// TIA Portal V21 export
FUNCTION "FC603" : Void   // FC603, LAD
TITLE = FC603
{ S7_Optimized_Access := 'TRUE' }
// CIP logic
// stored: AutoNumber false, SetENOAutomatically false
   VAR_TEMP
      temp : Int;
      re : Bool;
   END_VAR
   VAR_TEMP   // added for the SCL form of the ladder/FBD networks
      _w1 : Bool;
      _w2 : Bool;
      _w3 : Bool;
   END_VAR
BEGIN

REGION Network 1: NoCycleSelectedInterlock
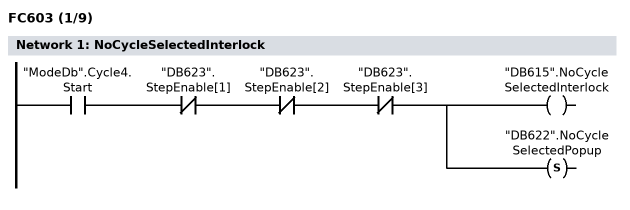
   RUNG wire#powerrail
      Contact( "ModeDb".Cycle4.Start )
      I_Contact( "DB623".StepEnable[1] )
      I_Contact( "DB623".StepEnable[2] )
      I_Contact( "DB623".StepEnable[3] )
      wire#w1
      Coil( "DB615".NoCycleSelectedInterlock )
   END_RUNG
   RUNG wire#w1
      S_Coil( "DB622".NoCycleSelectedPopup )
   END_RUNG
   // the same network as SCL:
   "DB615".NoCycleSelectedInterlock := "ModeDb".Cycle4.Start AND NOT "DB623".StepEnable[1] AND NOT "DB623".StepEnable[2] AND NOT "DB623".StepEnable[3];
   IF "DB615".NoCycleSelectedInterlock THEN "DB622".NoCycleSelectedPopup := TRUE; END_IF;
END_REGION

REGION Network 2: "DB615".Fault
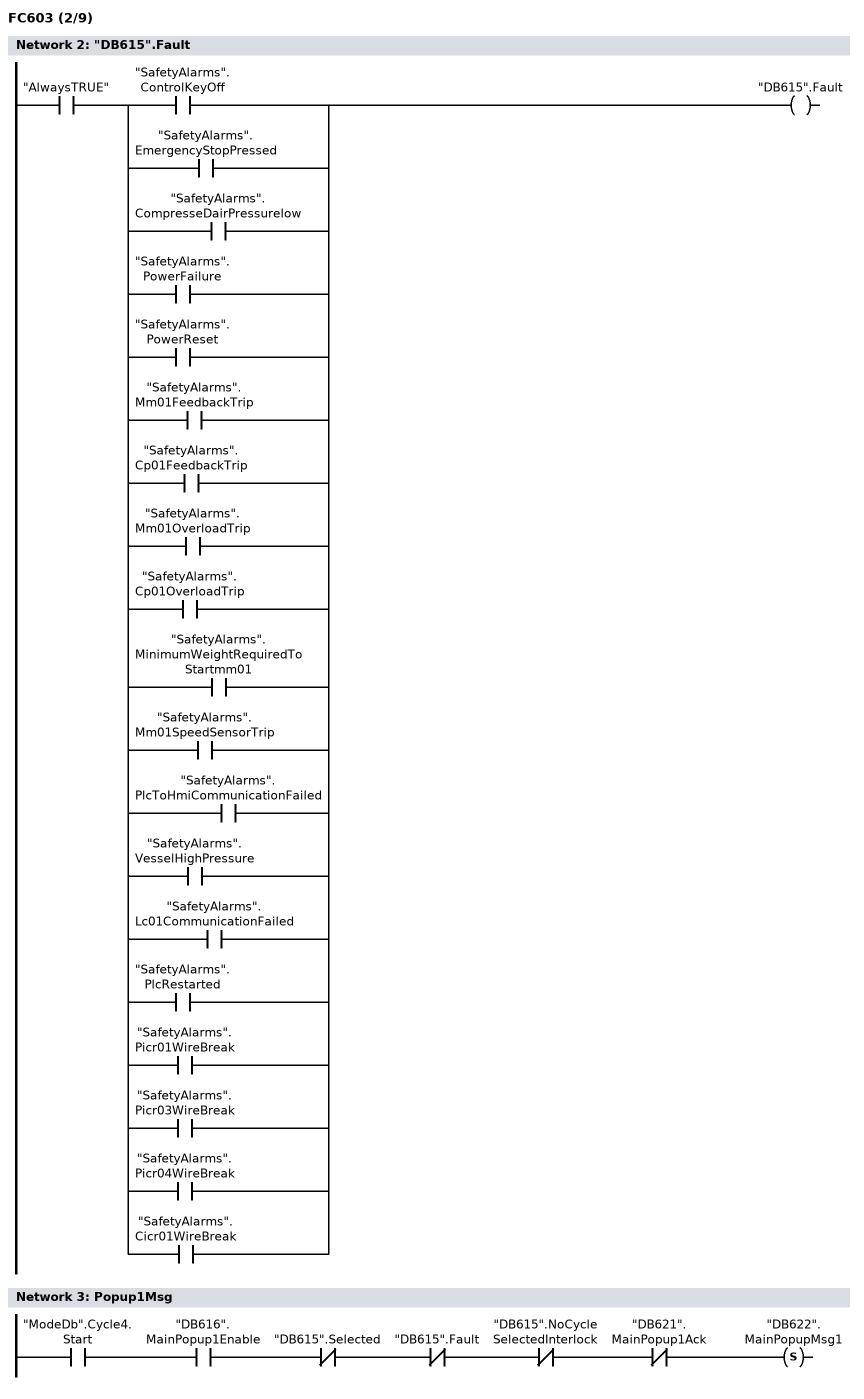
   RUNG wire#powerrail
      Contact( "AlwaysTRUE" )
      wire#w1
      Contact( "SafetyAlarms".ControlKeyOff )
      wire#w2
      Coil( "DB615".Fault )
   END_RUNG
   RUNG wire#w1
      Contact( "SafetyAlarms".EmergencyStopPressed )
   END_RUNG wire#w2
   RUNG wire#w1
      Contact( "SafetyAlarms".CompresseDairPressurelow )
   END_RUNG wire#w2
   RUNG wire#w1
      Contact( "SafetyAlarms".PowerFailure )
   END_RUNG wire#w2
   RUNG wire#w1
      Contact( "SafetyAlarms".PowerReset )
   END_RUNG wire#w2
   RUNG wire#w1
      Contact( "SafetyAlarms".Mm01FeedbackTrip )
   END_RUNG wire#w2
   RUNG wire#w1
      Contact( "SafetyAlarms".Cp01FeedbackTrip )
   END_RUNG wire#w2
   RUNG wire#w1
      Contact( "SafetyAlarms".Mm01OverloadTrip )
   END_RUNG wire#w2
   RUNG wire#w1
      Contact( "SafetyAlarms".Cp01OverloadTrip )
   END_RUNG wire#w2
   RUNG wire#w1
      Contact( "SafetyAlarms".MinimumWeightRequiredToStartmm01 )
   END_RUNG wire#w2
   RUNG wire#w1
      Contact( "SafetyAlarms".Mm01SpeedSensorTrip )
   END_RUNG wire#w2
   RUNG wire#w1
      Contact( "SafetyAlarms".PlcToHmiCommunicationFailed )
   END_RUNG wire#w2
   RUNG wire#w1
      Contact( "SafetyAlarms".VesselHighPressure )
   END_RUNG wire#w2
   RUNG wire#w1
      Contact( "SafetyAlarms".Lc01CommunicationFailed )
   END_RUNG wire#w2
   RUNG wire#w1
      Contact( "SafetyAlarms".PlcRestarted )
   END_RUNG wire#w2
   RUNG wire#w1
      Contact( "SafetyAlarms".Picr01WireBreak )
   END_RUNG wire#w2
   RUNG wire#w1
      Contact( "SafetyAlarms".Picr03WireBreak )
   END_RUNG wire#w2
   RUNG wire#w1
      Contact( "SafetyAlarms".Picr04WireBreak )
   END_RUNG wire#w2
   RUNG wire#w1
      Contact( "SafetyAlarms".Cicr01WireBreak )
   END_RUNG wire#w2
   // the same network as SCL:
   "DB615".Fault := "AlwaysTRUE" AND ("SafetyAlarms".ControlKeyOff OR "SafetyAlarms".EmergencyStopPressed OR "SafetyAlarms".CompresseDairPressurelow OR "SafetyAlarms".PowerFailure OR "SafetyAlarms".PowerReset OR "SafetyAlarms".Mm01FeedbackTrip OR "SafetyAlarms".Cp01FeedbackTrip OR "SafetyAlarms".Mm01OverloadTrip OR "SafetyAlarms".Cp01OverloadTrip OR "SafetyAlarms".MinimumWeightRequiredToStartmm01 OR "SafetyAlarms".Mm01SpeedSensorTrip OR "SafetyAlarms".PlcToHmiCommunicationFailed OR "SafetyAlarms".VesselHighPressure OR "SafetyAlarms".Lc01CommunicationFailed OR "SafetyAlarms".PlcRestarted OR "SafetyAlarms".Picr01WireBreak OR "SafetyAlarms".Picr03WireBreak OR "SafetyAlarms".Picr04WireBreak OR "SafetyAlarms".Cicr01WireBreak);
END_REGION

REGION Network 3: Popup1Msg
   RUNG wire#powerrail
      Contact( "ModeDb".Cycle4.Start )
      Contact( "DB616".MainPopup1Enable )
      I_Contact( "DB615".Selected )
      I_Contact( "DB615".Fault )
      I_Contact( "DB615".NoCycleSelectedInterlock )
      I_Contact( "DB621".MainPopup1Ack )
      S_Coil( "DB622".MainPopupMsg1 )
   END_RUNG
   // the same network as SCL:
   IF "ModeDb".Cycle4.Start AND "DB616".MainPopup1Enable AND NOT "DB615".Selected AND NOT "DB615".Fault AND NOT "DB615".NoCycleSelectedInterlock AND NOT "DB621".MainPopup1Ack THEN
       "DB622".MainPopupMsg1 := TRUE;
   END_IF;
END_REGION

REGION Network 4: Popup2Msg
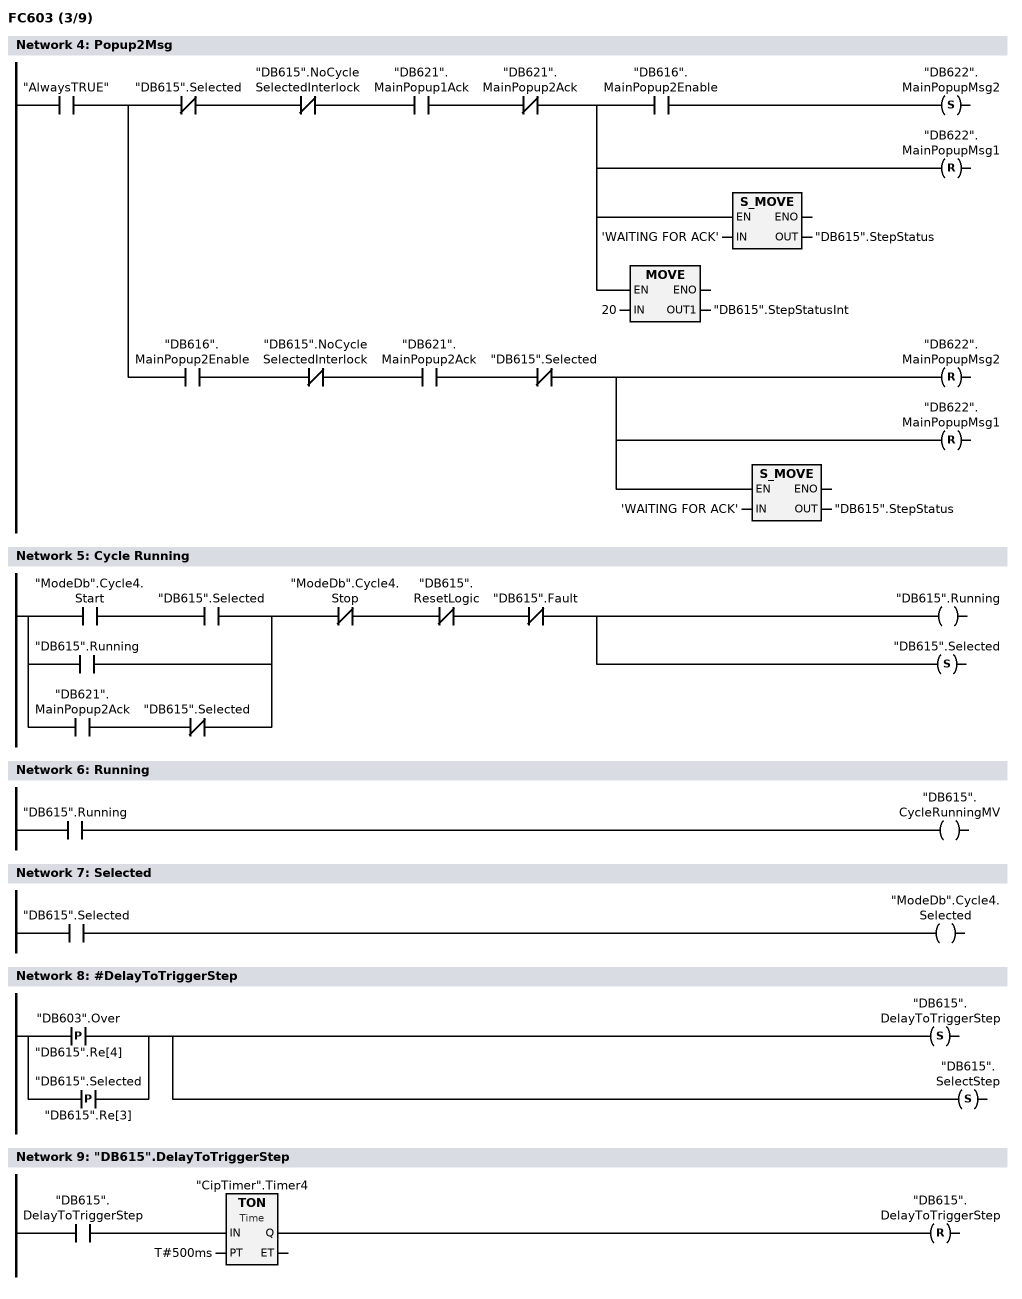
   RUNG wire#powerrail
      Contact( "AlwaysTRUE" )
      wire#w1
      I_Contact( "DB615".Selected )
      I_Contact( "DB615".NoCycleSelectedInterlock )
      Contact( "DB621".MainPopup1Ack )
      I_Contact( "DB621".MainPopup2Ack )
      wire#w2
      Contact( "DB616".MainPopup2Enable )
      S_Coil( "DB622".MainPopupMsg2 )
   END_RUNG
   RUNG wire#w2
      R_Coil( "DB622".MainPopupMsg1 )
   END_RUNG
   RUNG wire#w2
      S_Move(in := 'WAITING FOR ACK', out => "DB615".StepStatus)
   END_RUNG
   RUNG wire#w2
      Move(in := 20, out1 => "DB615".StepStatusInt)
   END_RUNG
   RUNG wire#w1
      Contact( "DB616".MainPopup2Enable )
      I_Contact( "DB615".NoCycleSelectedInterlock )
      Contact( "DB621".MainPopup2Ack )
      I_Contact( "DB615".Selected )
      wire#w3
      R_Coil( "DB622".MainPopupMsg2 )
   END_RUNG
   RUNG wire#w3
      R_Coil( "DB622".MainPopupMsg1 )
   END_RUNG
   RUNG wire#w3
      S_Move(in := 'WAITING FOR ACK', out => "DB615".StepStatus)
   END_RUNG
   // the same network as SCL:
   #_w1 := "AlwaysTRUE" AND NOT "DB615".Selected AND NOT "DB615".NoCycleSelectedInterlock AND "DB621".MainPopup1Ack AND NOT "DB621".MainPopup2Ack;
   IF #_w1 AND "DB616".MainPopup2Enable THEN "DB622".MainPopupMsg2 := TRUE; END_IF;
   IF #_w1 THEN
       "DB622".MainPopupMsg1 := FALSE;
       "DB615".StepStatus := 'WAITING FOR ACK';
       "DB615".StepStatusInt := 20;
   END_IF;
   IF "AlwaysTRUE" AND "DB616".MainPopup2Enable AND NOT "DB615".NoCycleSelectedInterlock AND "DB621".MainPopup2Ack AND NOT "DB615".Selected THEN
       "DB622".MainPopupMsg2 := FALSE;
       "DB622".MainPopupMsg1 := FALSE;
       "DB615".StepStatus := 'WAITING FOR ACK';
   END_IF;
END_REGION

REGION Network 5: Cycle Running
   RUNG wire#powerrail
      Contact( "ModeDb".Cycle4.Start )
      Contact( "DB615".Selected )
      wire#w1
      I_Contact( "ModeDb".Cycle4.Stop )
      I_Contact( "DB615".ResetLogic )
      I_Contact( "DB615".Fault )
      wire#w2
      Coil( "DB615".Running )
   END_RUNG
   RUNG wire#powerrail
      Contact( "DB615".Running )
   END_RUNG wire#w1
   RUNG wire#powerrail
      Contact( "DB621".MainPopup2Ack )
      I_Contact( "DB615".Selected )
   END_RUNG wire#w1
   RUNG wire#w2
      S_Coil( "DB615".Selected )
   END_RUNG
   // the same network as SCL:
   "DB615".Running := (("ModeDb".Cycle4.Start AND "DB615".Selected) OR "DB615".Running OR ("DB621".MainPopup2Ack AND NOT "DB615".Selected)) AND NOT "ModeDb".Cycle4.Stop AND NOT "DB615".ResetLogic AND NOT "DB615".Fault;
   IF "DB615".Running THEN "DB615".Selected := TRUE; END_IF;
END_REGION

REGION Network 6: Running
   RUNG wire#powerrail
      Contact( "DB615".Running )
      Coil( "DB615".CycleRunningMV )
   END_RUNG
   // the same network as SCL:
   "DB615".CycleRunningMV := "DB615".Running;
END_REGION

REGION Network 7: Selected
   RUNG wire#powerrail
      Contact( "DB615".Selected )
      Coil( "ModeDb".Cycle4.Selected )
   END_RUNG
   // the same network as SCL:
   "ModeDb".Cycle4.Selected := "DB615".Selected;
END_REGION

REGION Network 8: #DelayToTriggerStep
   RUNG wire#powerrail
      P_Contact(operand := "DB603".Over, bit := "DB615".Re[4])
      wire#w1
      S_Coil( "DB615".DelayToTriggerStep )
   END_RUNG
   RUNG wire#powerrail
      P_Contact(operand := "DB615".Selected, bit := "DB615".Re[3])
   END_RUNG wire#w1
   RUNG wire#w1
      S_Coil( "DB615".SelectStep )
   END_RUNG
   // the same network as SCL:
   #_w1 := "DB603".Over AND NOT "DB615".Re[4];   // rising edge of "DB603".Over
   "DB615".Re[4] := "DB603".Over;
   #_w2 := "DB615".Selected AND NOT "DB615".Re[3];   // rising edge of "DB615".Selected
   "DB615".Re[3] := "DB615".Selected;
   IF #_w1 OR #_w2 THEN
       "DB615".DelayToTriggerStep := TRUE;
       "DB615".SelectStep := TRUE;
   END_IF;
END_REGION

REGION Network 9: "DB615".DelayToTriggerStep
   RUNG wire#powerrail
      Contact( "DB615".DelayToTriggerStep )
      { S7_Templates := "time_type := Time" } "CipTimer".Timer4.TON(pt := T#500ms, et =>)
      R_Coil( "DB615".DelayToTriggerStep )
   END_RUNG
   // the same network as SCL:
   "CipTimer".Timer4.TON(IN := "DB615".DelayToTriggerStep, PT := T#500ms);
   IF "CipTimer".Timer4.Q THEN "DB615".DelayToTriggerStep := FALSE; END_IF;
END_REGION

REGION Network 10: CYCLE STATUS
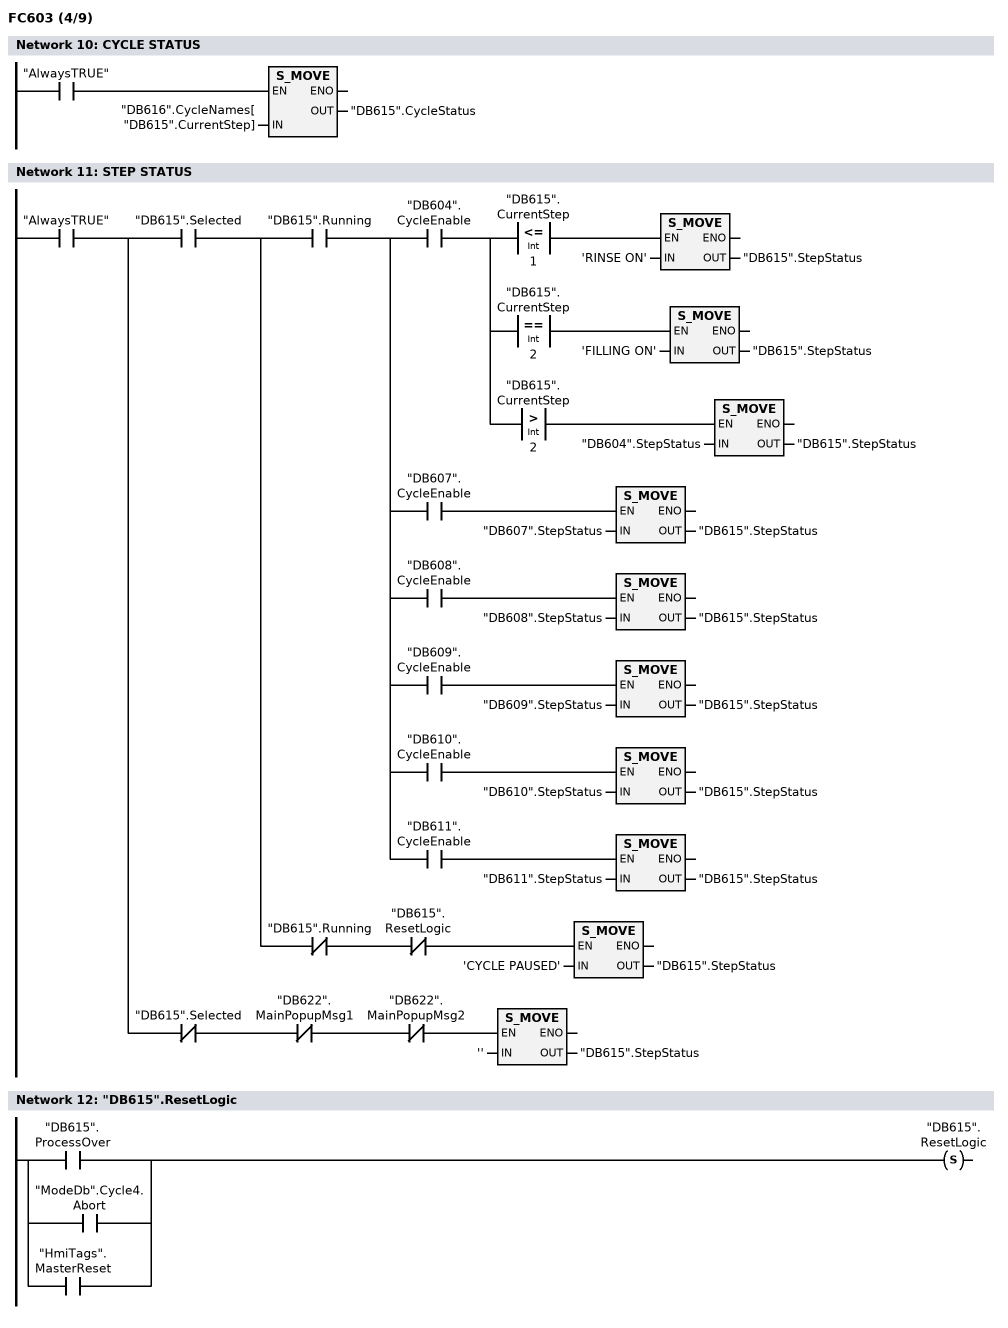
   RUNG wire#powerrail
      Contact( "AlwaysTRUE" )
      S_Move(in := "DB616".CycleNames["DB615".CurrentStep], out => "DB615".CycleStatus)
   END_RUNG
   // the same network as SCL:
   IF "AlwaysTRUE" THEN "DB615".CycleStatus := "DB616".CycleNames["DB615".CurrentStep]; END_IF;
END_REGION

REGION Network 11: STEP STATUS
   RUNG wire#powerrail
      Contact( "AlwaysTRUE" )
      wire#w1
      Contact( "DB615".Selected )
      wire#w2
      Contact( "DB615".Running )
      wire#w3
      Contact( "DB604".CycleEnable )
      wire#w4
      { S7_Templates := "SrcType := Int" } LE_Contact(in1 := "DB615".CurrentStep, in2 := 1)
      S_Move(in := 'RINSE ON', out => "DB615".StepStatus)
   END_RUNG
   RUNG wire#w4
      { S7_Templates := "SrcType := Int" } EQ_Contact(in1 := "DB615".CurrentStep, in2 := 2)
      S_Move(in := 'FILLING ON', out => "DB615".StepStatus)
   END_RUNG
   RUNG wire#w4
      { S7_Templates := "SrcType := Int" } GT_Contact(in1 := "DB615".CurrentStep, in2 := 2)
      S_Move(in := "DB604".StepStatus, out => "DB615".StepStatus)
   END_RUNG
   RUNG wire#w3
      Contact( "DB607".CycleEnable )
      S_Move(in := "DB607".StepStatus, out => "DB615".StepStatus)
   END_RUNG
   RUNG wire#w3
      Contact( "DB608".CycleEnable )
      S_Move(in := "DB608".StepStatus, out => "DB615".StepStatus)
   END_RUNG
   RUNG wire#w3
      Contact( "DB609".CycleEnable )
      S_Move(in := "DB609".StepStatus, out => "DB615".StepStatus)
   END_RUNG
   RUNG wire#w3
      Contact( "DB610".CycleEnable )
      S_Move(in := "DB610".StepStatus, out => "DB615".StepStatus)
   END_RUNG
   RUNG wire#w3
      Contact( "DB611".CycleEnable )
      S_Move(in := "DB611".StepStatus, out => "DB615".StepStatus)
   END_RUNG
   RUNG wire#w2
      I_Contact( "DB615".Running )
      I_Contact( "DB615".ResetLogic )
      S_Move(in := 'CYCLE PAUSED', out => "DB615".StepStatus)
   END_RUNG
   RUNG wire#w1
      I_Contact( "DB615".Selected )
      I_Contact( "DB622".MainPopupMsg1 )
      I_Contact( "DB622".MainPopupMsg2 )
      S_Move(in := '', out => "DB615".StepStatus)
   END_RUNG
   // the same network as SCL:
   #_w1 := "AlwaysTRUE" AND "DB615".Selected;
   #_w2 := #_w1 AND "DB615".Running;
   #_w3 := #_w2 AND "DB604".CycleEnable;
   IF #_w3 AND ("DB615".CurrentStep <= 1) THEN "DB615".StepStatus := 'RINSE ON'; END_IF;
   IF #_w3 AND ("DB615".CurrentStep = 2) THEN "DB615".StepStatus := 'FILLING ON'; END_IF;
   IF #_w3 AND ("DB615".CurrentStep > 2) THEN "DB615".StepStatus := "DB604".StepStatus; END_IF;
   IF #_w2 AND "DB607".CycleEnable THEN "DB615".StepStatus := "DB607".StepStatus; END_IF;
   IF #_w2 AND "DB608".CycleEnable THEN "DB615".StepStatus := "DB608".StepStatus; END_IF;
   IF #_w2 AND "DB609".CycleEnable THEN "DB615".StepStatus := "DB609".StepStatus; END_IF;
   IF #_w2 AND "DB610".CycleEnable THEN "DB615".StepStatus := "DB610".StepStatus; END_IF;
   IF #_w2 AND "DB611".CycleEnable THEN "DB615".StepStatus := "DB611".StepStatus; END_IF;
   IF #_w1 AND NOT "DB615".Running AND NOT "DB615".ResetLogic THEN
       "DB615".StepStatus := 'CYCLE PAUSED';
   END_IF;
   IF "AlwaysTRUE" AND NOT "DB615".Selected AND NOT "DB622".MainPopupMsg1 AND NOT "DB622".MainPopupMsg2 THEN
       "DB615".StepStatus := '';
   END_IF;
END_REGION

REGION Network 12: "DB615".ResetLogic
   RUNG wire#powerrail
      Contact( "DB615".ProcessOver )
      wire#w1
      S_Coil( "DB615".ResetLogic )
   END_RUNG
   RUNG wire#powerrail
      Contact( "ModeDb".Cycle4.Abort )
   END_RUNG wire#w1
   RUNG wire#powerrail
      Contact( "HmiTags".MasterReset )
   END_RUNG wire#w1
   // the same network as SCL:
   IF "DB615".ProcessOver OR "ModeDb".Cycle4.Abort OR "HmiTags".MasterReset THEN
       "DB615".ResetLogic := TRUE;
   END_IF;
END_REGION

REGION Network 13: "Printing".ResultCip
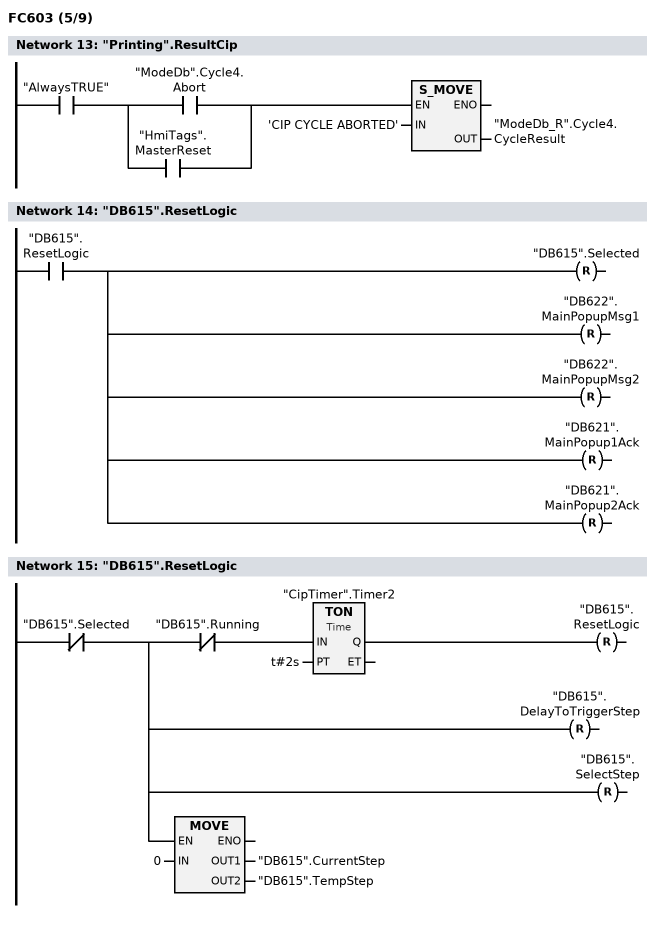
   RUNG wire#powerrail
      Contact( "AlwaysTRUE" )
      wire#w1
      Contact( "ModeDb".Cycle4.Abort )
      wire#w2
      S_Move(in := 'CIP CYCLE ABORTED', out => "ModeDb_R".Cycle4.CycleResult)
   END_RUNG
   RUNG wire#w1
      Contact( "HmiTags".MasterReset )
   END_RUNG wire#w2
   // the same network as SCL:
   IF "AlwaysTRUE" AND ("ModeDb".Cycle4.Abort OR "HmiTags".MasterReset) THEN
       "ModeDb_R".Cycle4.CycleResult := 'CIP CYCLE ABORTED';
   END_IF;
END_REGION

REGION Network 14: "DB615".ResetLogic
   RUNG wire#powerrail
      Contact( "DB615".ResetLogic )
      wire#w1
      R_Coil( "DB615".Selected )
   END_RUNG
   RUNG wire#w1
      R_Coil( "DB622".MainPopupMsg1 )
   END_RUNG
   RUNG wire#w1
      R_Coil( "DB622".MainPopupMsg2 )
   END_RUNG
   RUNG wire#w1
      R_Coil( "DB621".MainPopup1Ack )
   END_RUNG
   RUNG wire#w1
      R_Coil( "DB621".MainPopup2Ack )
   END_RUNG
   // the same network as SCL:
   IF "DB615".ResetLogic THEN
       "DB615".Selected := FALSE;
       "DB622".MainPopupMsg1 := FALSE;
       "DB622".MainPopupMsg2 := FALSE;
       "DB621".MainPopup1Ack := FALSE;
       "DB621".MainPopup2Ack := FALSE;
   END_IF;
END_REGION

REGION Network 15: "DB615".ResetLogic
   RUNG wire#powerrail
      I_Contact( "DB615".Selected )
      wire#w1
      I_Contact( "DB615".Running )
      { S7_Templates := "time_type := Time" } "CipTimer".Timer2.TON(pt := t#2s, et =>)
      R_Coil( "DB615".ResetLogic )
   END_RUNG
   RUNG wire#w1
      R_Coil( "DB615".DelayToTriggerStep )
   END_RUNG
   RUNG wire#w1
      R_Coil( "DB615".SelectStep )
   END_RUNG
   RUNG wire#w1
      Move(in := 0, out1 => "DB615".CurrentStep, out2 => "DB615".TempStep)
   END_RUNG
   // the same network as SCL:
   "CipTimer".Timer2.TON(IN := NOT "DB615".Selected AND NOT "DB615".Running, PT := t#2s);
   IF "CipTimer".Timer2.Q THEN "DB615".ResetLogic := FALSE; END_IF;
   IF NOT "DB615".Selected THEN
       "DB615".DelayToTriggerStep := FALSE;
       "DB615".SelectStep := FALSE;
       "DB615".CurrentStep := 0;
       "DB615".TempStep := 0;
   END_IF;
END_REGION

REGION Network 16: Button Reset
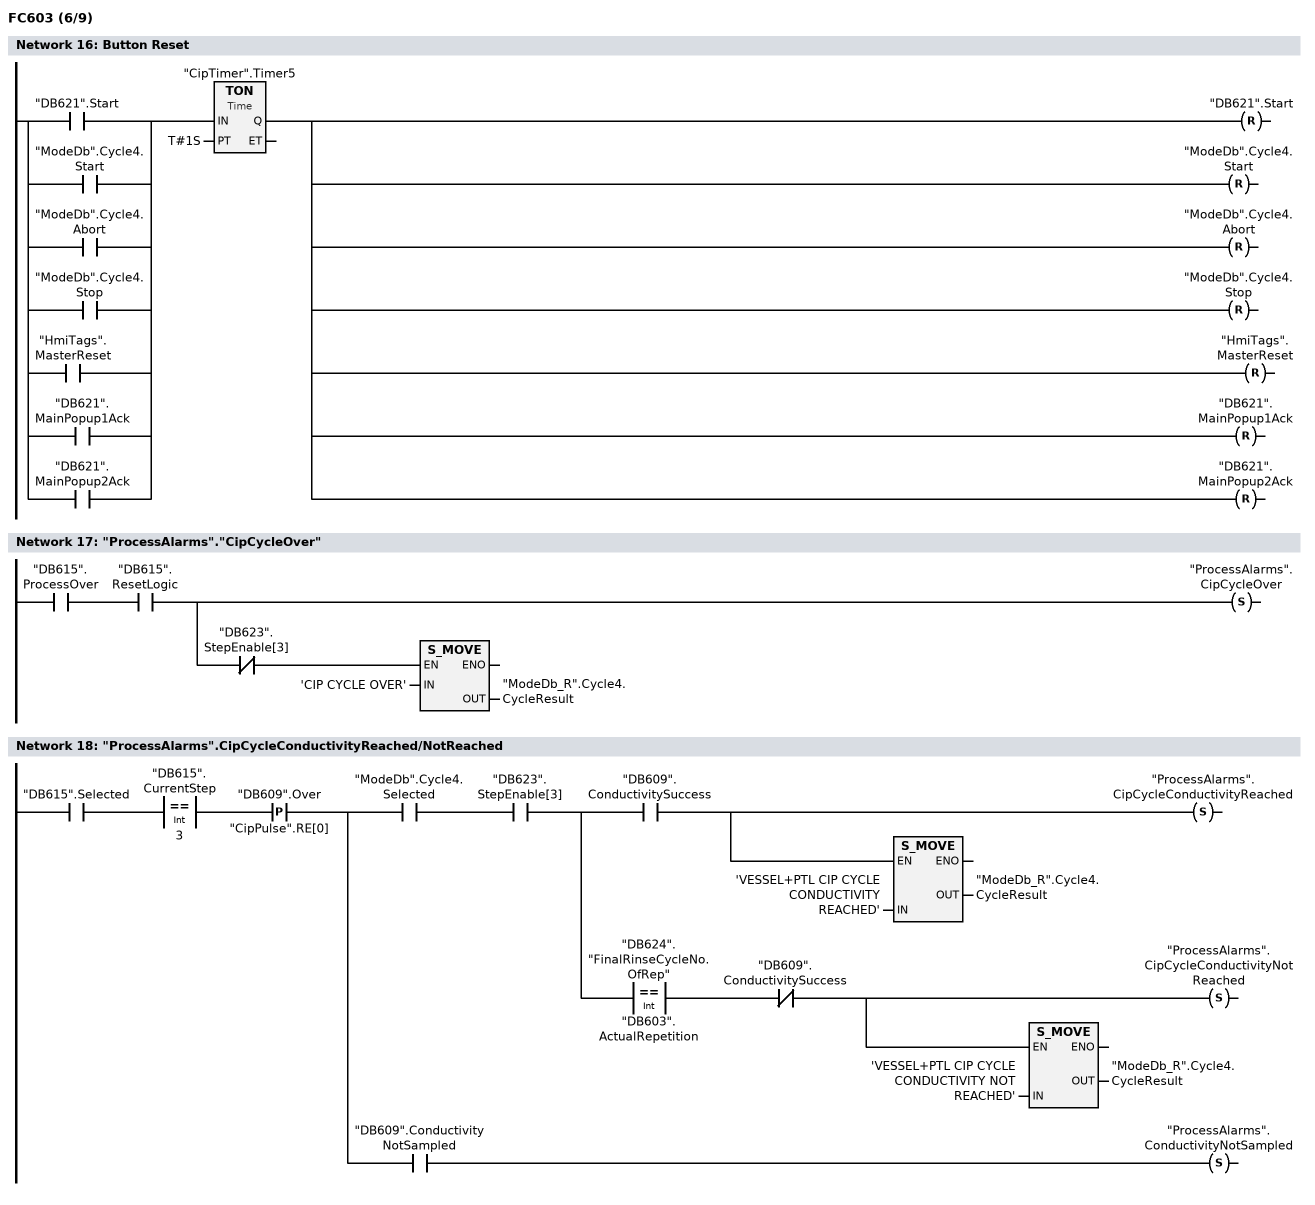
   RUNG wire#powerrail
      Contact( "DB621".Start )
      wire#w1
      { S7_Templates := "time_type := Time" } "CipTimer".Timer5.TON(pt := T#1S, et =>)
      wire#w2
      R_Coil( "DB621".Start )
   END_RUNG
   RUNG wire#powerrail
      Contact( "ModeDb".Cycle4.Start )
   END_RUNG wire#w1
   RUNG wire#powerrail
      Contact( "ModeDb".Cycle4.Abort )
   END_RUNG wire#w1
   RUNG wire#powerrail
      Contact( "ModeDb".Cycle4.Stop )
   END_RUNG wire#w1
   RUNG wire#powerrail
      Contact( "HmiTags".MasterReset )
   END_RUNG wire#w1
   RUNG wire#powerrail
      Contact( "DB621".MainPopup1Ack )
   END_RUNG wire#w1
   RUNG wire#powerrail
      Contact( "DB621".MainPopup2Ack )
   END_RUNG wire#w1
   RUNG wire#w2
      R_Coil( "ModeDb".Cycle4.Start )
   END_RUNG
   RUNG wire#w2
      R_Coil( "ModeDb".Cycle4.Abort )
   END_RUNG
   RUNG wire#w2
      R_Coil( "ModeDb".Cycle4.Stop )
   END_RUNG
   RUNG wire#w2
      R_Coil( "HmiTags".MasterReset )
   END_RUNG
   RUNG wire#w2
      R_Coil( "DB621".MainPopup1Ack )
   END_RUNG
   RUNG wire#w2
      R_Coil( "DB621".MainPopup2Ack )
   END_RUNG
   // the same network as SCL:
   "CipTimer".Timer5.TON(IN := "DB621".Start OR "ModeDb".Cycle4.Start OR "ModeDb".Cycle4.Abort OR "ModeDb".Cycle4.Stop OR "HmiTags".MasterReset OR "DB621".MainPopup1Ack OR "DB621".MainPopup2Ack,
                         PT := T#1S);
   IF "CipTimer".Timer5.Q THEN
       "DB621".Start := FALSE;
       "ModeDb".Cycle4.Start := FALSE;
       "ModeDb".Cycle4.Abort := FALSE;
       "ModeDb".Cycle4.Stop := FALSE;
       "HmiTags".MasterReset := FALSE;
       "DB621".MainPopup1Ack := FALSE;
       "DB621".MainPopup2Ack := FALSE;
   END_IF;
END_REGION

REGION Network 17: "ProcessAlarms"."CipCycleOver"
   RUNG wire#powerrail
      Contact( "DB615".ProcessOver )
      Contact( "DB615".ResetLogic )
      wire#w1
      S_Coil( "ProcessAlarms".CipCycleOver )
   END_RUNG
   RUNG wire#w1
      I_Contact( "DB623".StepEnable[3] )
      S_Move(in := 'CIP CYCLE OVER', out => "ModeDb_R".Cycle4.CycleResult)
   END_RUNG
   // the same network as SCL:
   #_w1 := "DB615".ProcessOver AND "DB615".ResetLogic;
   IF #_w1 THEN "ProcessAlarms".CipCycleOver := TRUE; END_IF;
   IF #_w1 AND NOT "DB623".StepEnable[3] THEN "ModeDb_R".Cycle4.CycleResult := 'CIP CYCLE OVER'; END_IF;
END_REGION

REGION Network 18: "ProcessAlarms".CipCycleConductivityReached/NotReached
   RUNG wire#powerrail
      Contact( "DB615".Selected )
      { S7_Templates := "SrcType := Int" } EQ_Contact(in1 := "DB615".CurrentStep, in2 := 3)
      P_Contact(operand := "DB609".Over, bit := "CipPulse".RE[0])
      wire#w1
      Contact( "ModeDb".Cycle4.Selected )
      Contact( "DB623".StepEnable[3] )
      wire#w2
      Contact( "DB609".ConductivitySuccess )
      wire#w3
      S_Coil( "ProcessAlarms".CipCycleConductivityReached )
   END_RUNG
   RUNG wire#w3
      S_Move(in := 'VESSEL+PTL CIP CYCLE CONDUCTIVITY REACHED', out => "ModeDb_R".Cycle4.CycleResult)
   END_RUNG
   RUNG wire#w2
      { S7_Templates := "SrcType := Int" } EQ_Contact(in1 := "DB624"."FinalRinseCycleNo.OfRep", in2 := "DB603".ActualRepetition)
      I_Contact( "DB609".ConductivitySuccess )
      wire#w4
      S_Coil( "ProcessAlarms".CipCycleConductivityNotReached )
   END_RUNG
   RUNG wire#w4
      S_Move(in := 'VESSEL+PTL CIP CYCLE CONDUCTIVITY NOT REACHED', out => "ModeDb_R".Cycle4.CycleResult)
   END_RUNG
   RUNG wire#w1
      Contact( "DB609".ConductivityNotSampled )
      S_Coil( "ProcessAlarms".ConductivityNotSampled )
   END_RUNG
   // the same network as SCL:
   #_w1 := "DB615".Selected AND ("DB615".CurrentStep = 3) AND "DB609".Over AND NOT "CipPulse".RE[0];   // rising edge of "DB609".Over
   "CipPulse".RE[0] := "DB609".Over;
   #_w2 := #_w1 AND "ModeDb".Cycle4.Selected AND "DB623".StepEnable[3];
   IF #_w2 AND "DB609".ConductivitySuccess THEN
       "ProcessAlarms".CipCycleConductivityReached := TRUE;
       "ModeDb_R".Cycle4.CycleResult := 'VESSEL+PTL CIP CYCLE CONDUCTIVITY REACHED';
   END_IF;
   IF #_w2 AND ("DB624"."FinalRinseCycleNo.OfRep" = "DB603".ActualRepetition) AND NOT "DB609".ConductivitySuccess THEN
       "ProcessAlarms".CipCycleConductivityNotReached := TRUE;
       "ModeDb_R".Cycle4.CycleResult := 'VESSEL+PTL CIP CYCLE CONDUCTIVITY NOT REACHED';
   END_IF;
   IF #_w1 AND "DB609".ConductivityNotSampled THEN "ProcessAlarms".ConductivityNotSampled := TRUE; END_IF;
END_REGION

REGION Network 19: "HmiTags".AlarmAck
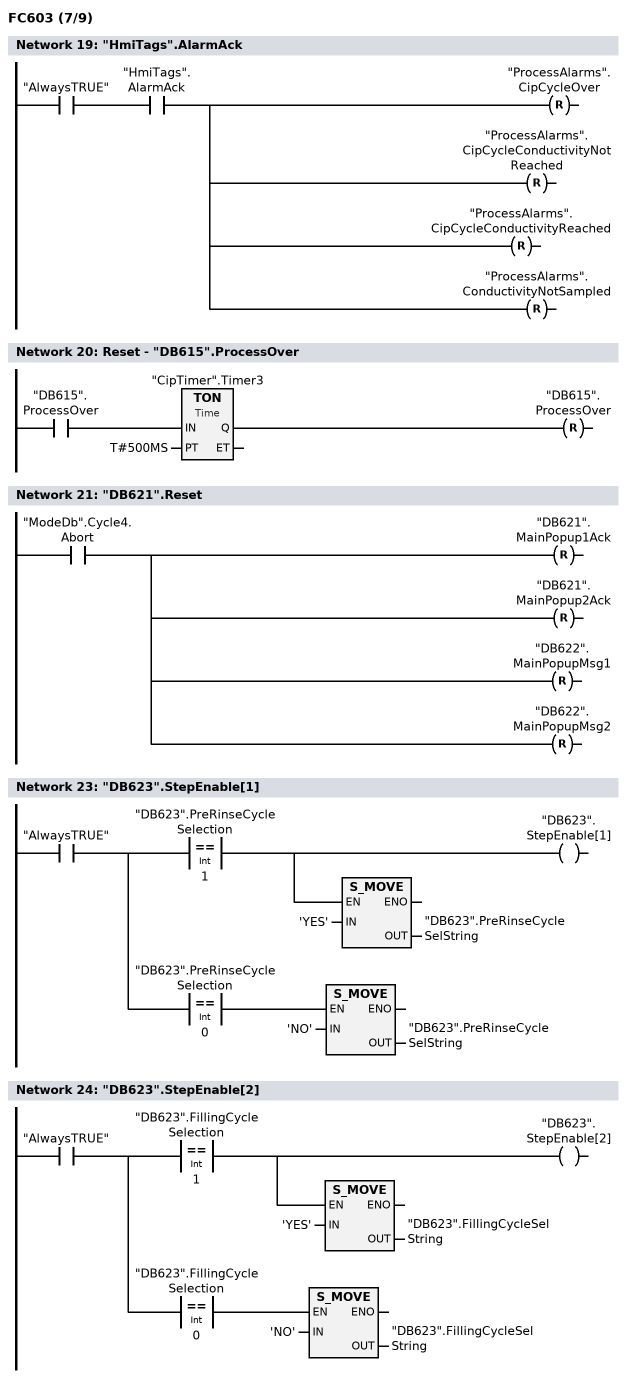
   RUNG wire#powerrail
      Contact( "AlwaysTRUE" )
      Contact( "HmiTags".AlarmAck )
      wire#w1
      R_Coil( "ProcessAlarms".CipCycleOver )
   END_RUNG
   RUNG wire#w1
      R_Coil( "ProcessAlarms".CipCycleConductivityNotReached )
   END_RUNG
   RUNG wire#w1
      R_Coil( "ProcessAlarms".CipCycleConductivityReached )
   END_RUNG
   RUNG wire#w1
      R_Coil( "ProcessAlarms".ConductivityNotSampled )
   END_RUNG
   // the same network as SCL:
   IF "AlwaysTRUE" AND "HmiTags".AlarmAck THEN
       "ProcessAlarms".CipCycleOver := FALSE;
       "ProcessAlarms".CipCycleConductivityNotReached := FALSE;
       "ProcessAlarms".CipCycleConductivityReached := FALSE;
       "ProcessAlarms".ConductivityNotSampled := FALSE;
   END_IF;
END_REGION

REGION Network 20: Reset - "DB615".ProcessOver
   RUNG wire#powerrail
      Contact( "DB615".ProcessOver )
      { S7_Templates := "time_type := Time" } "CipTimer".Timer3.TON(pt := T#500MS, et =>)
      R_Coil( "DB615".ProcessOver )
   END_RUNG
   // the same network as SCL:
   "CipTimer".Timer3.TON(IN := "DB615".ProcessOver, PT := T#500MS);
   IF "CipTimer".Timer3.Q THEN "DB615".ProcessOver := FALSE; END_IF;
END_REGION

REGION Network 21: "DB621".Reset
   RUNG wire#powerrail
      Contact( "ModeDb".Cycle4.Abort )
      wire#w1
      R_Coil( "DB621".MainPopup1Ack )
   END_RUNG
   RUNG wire#w1
      R_Coil( "DB621".MainPopup2Ack )
   END_RUNG
   RUNG wire#w1
      R_Coil( "DB622".MainPopupMsg1 )
   END_RUNG
   RUNG wire#w1
      R_Coil( "DB622".MainPopupMsg2 )
   END_RUNG
   // the same network as SCL:
   IF "ModeDb".Cycle4.Abort THEN
       "DB621".MainPopup1Ack := FALSE;
       "DB621".MainPopup2Ack := FALSE;
       "DB622".MainPopupMsg1 := FALSE;
       "DB622".MainPopupMsg2 := FALSE;
   END_IF;
END_REGION

REGION Network 22: *********MV 3000 *****************
END_REGION

REGION Network 23: "DB623".StepEnable[1]
   RUNG wire#powerrail
      Contact( "AlwaysTRUE" )
      wire#w1
      { S7_Templates := "SrcType := Int" } EQ_Contact(in1 := "DB623".PreRinseCycleSelection, in2 := 1)
      wire#w2
      Coil( "DB623".StepEnable[1] )
   END_RUNG
   RUNG wire#w2
      S_Move(in := 'YES', out => "DB623".PreRinseCycleSelString)
   END_RUNG
   RUNG wire#w1
      { S7_Templates := "SrcType := Int" } EQ_Contact(in1 := "DB623".PreRinseCycleSelection, in2 := 0)
      S_Move(in := 'NO', out => "DB623".PreRinseCycleSelString)
   END_RUNG
   // the same network as SCL:
   "DB623".StepEnable[1] := "AlwaysTRUE" AND ("DB623".PreRinseCycleSelection = 1);
   IF "AlwaysTRUE" AND ("DB623".PreRinseCycleSelection = 1) THEN
       "DB623".PreRinseCycleSelString := 'YES';
   END_IF;
   IF "AlwaysTRUE" AND ("DB623".PreRinseCycleSelection = 0) THEN
       "DB623".PreRinseCycleSelString := 'NO';
   END_IF;
END_REGION

REGION Network 24: "DB623".StepEnable[2]
   RUNG wire#powerrail
      Contact( "AlwaysTRUE" )
      wire#w1
      { S7_Templates := "SrcType := Int" } EQ_Contact(in1 := "DB623".FillingCycleSelection, in2 := 1)
      wire#w2
      Coil( "DB623".StepEnable[2] )
   END_RUNG
   RUNG wire#w2
      S_Move(in := 'YES', out => "DB623".FillingCycleSelString)
   END_RUNG
   RUNG wire#w1
      { S7_Templates := "SrcType := Int" } EQ_Contact(in1 := "DB623".FillingCycleSelection, in2 := 0)
      S_Move(in := 'NO', out => "DB623".FillingCycleSelString)
   END_RUNG
   // the same network as SCL:
   "DB623".StepEnable[2] := "AlwaysTRUE" AND ("DB623".FillingCycleSelection = 1);
   IF "AlwaysTRUE" AND ("DB623".FillingCycleSelection = 1) THEN
       "DB623".FillingCycleSelString := 'YES';
   END_IF;
   IF "AlwaysTRUE" AND ("DB623".FillingCycleSelection = 0) THEN
       "DB623".FillingCycleSelString := 'NO';
   END_IF;
END_REGION

REGION Network 25: "DB623".StepEnable[3]
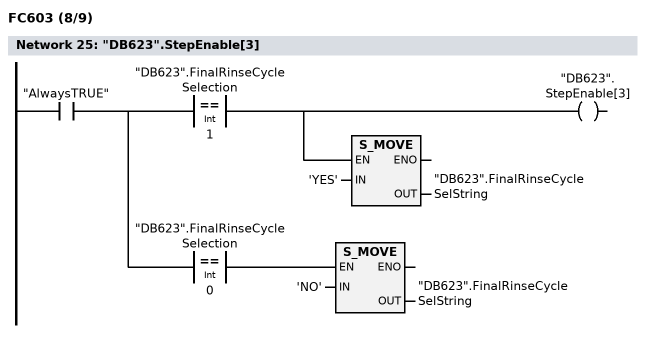
   RUNG wire#powerrail
      Contact( "AlwaysTRUE" )
      wire#w1
      { S7_Templates := "SrcType := Int" } EQ_Contact(in1 := "DB623".FinalRinseCycleSelection, in2 := 1)
      wire#w2
      Coil( "DB623".StepEnable[3] )
   END_RUNG
   RUNG wire#w2
      S_Move(in := 'YES', out => "DB623".FinalRinseCycleSelString)
   END_RUNG
   RUNG wire#w1
      { S7_Templates := "SrcType := Int" } EQ_Contact(in1 := "DB623".FinalRinseCycleSelection, in2 := 0)
      S_Move(in := 'NO', out => "DB623".FinalRinseCycleSelString)
   END_RUNG
   // the same network as SCL:
   "DB623".StepEnable[3] := "AlwaysTRUE" AND ("DB623".FinalRinseCycleSelection = 1);
   IF "AlwaysTRUE" AND ("DB623".FinalRinseCycleSelection = 1) THEN
       "DB623".FinalRinseCycleSelString := 'YES';
   END_IF;
   IF "AlwaysTRUE" AND ("DB623".FinalRinseCycleSelection = 0) THEN
       "DB623".FinalRinseCycleSelString := 'NO';
   END_IF;
END_REGION

REGION Network 27: Para Passing of AP AI sensor
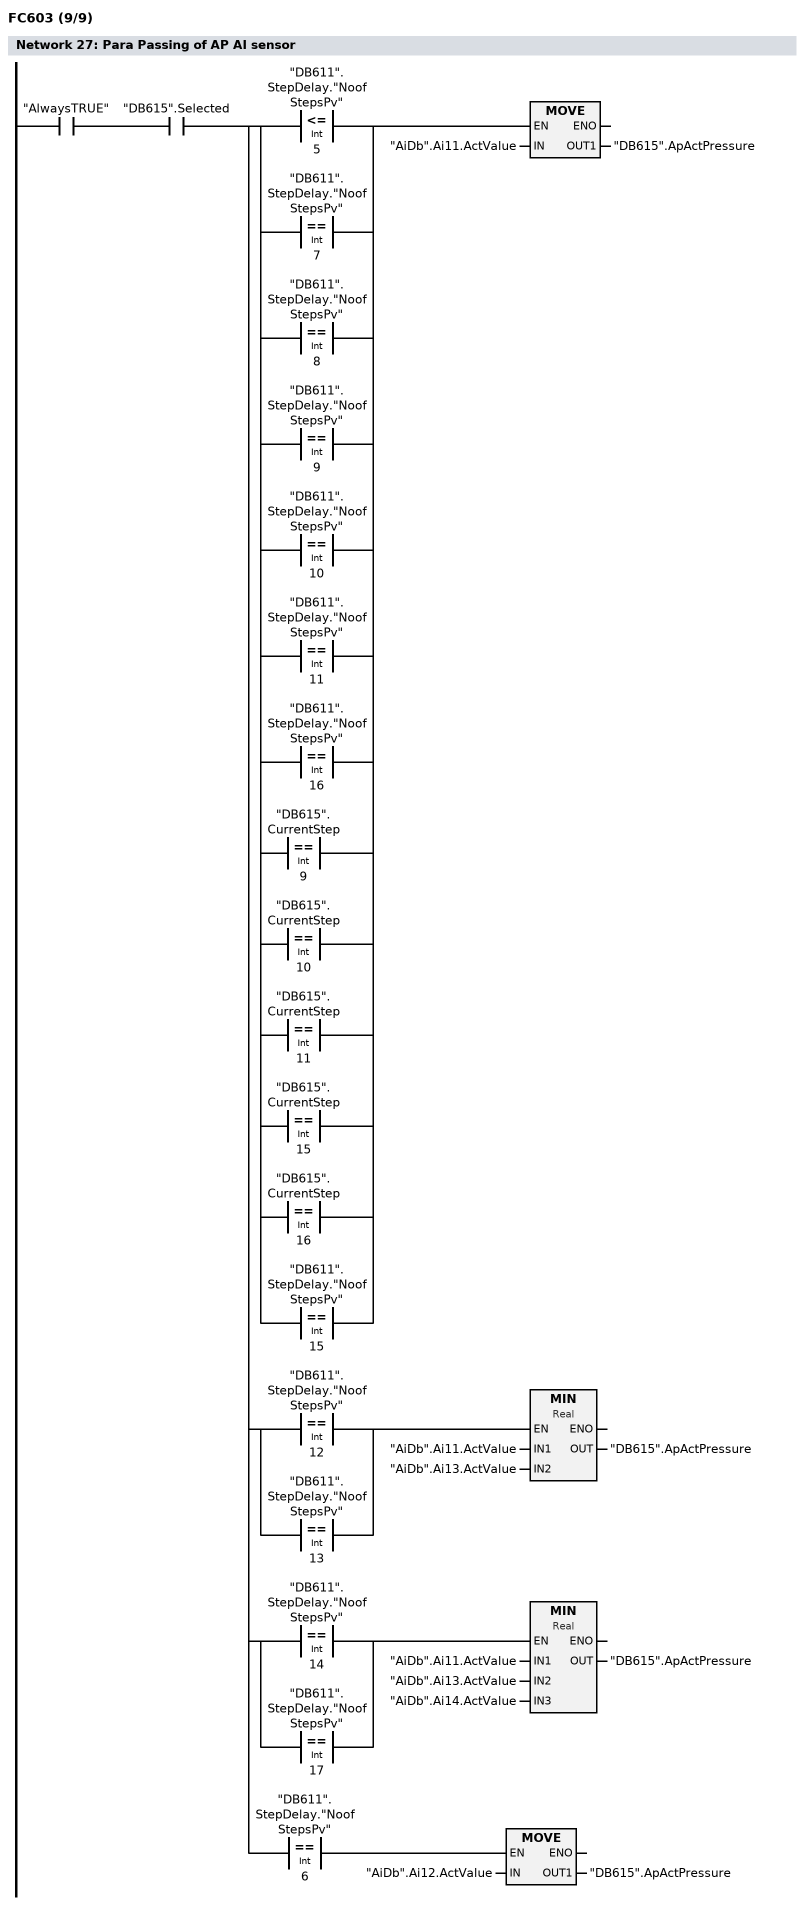
   RUNG wire#powerrail
      Contact( "AlwaysTRUE" )
      Contact( "DB615".Selected )
      wire#w1
      { S7_Templates := "SrcType := Int" } LE_Contact(in1 := "DB611".StepDelay."Noof StepsPv", in2 := 5)
      wire#w2
      Move(in := "AiDb".Ai11.ActValue, out1 => "DB615".ApActPressure)
   END_RUNG
   RUNG wire#w1
      { S7_Templates := "SrcType := Int" } EQ_Contact(in1 := "DB611".StepDelay."Noof StepsPv", in2 := 7)
   END_RUNG wire#w2
   RUNG wire#w1
      { S7_Templates := "SrcType := Int" } EQ_Contact(in1 := "DB611".StepDelay."Noof StepsPv", in2 := 8)
   END_RUNG wire#w2
   RUNG wire#w1
      { S7_Templates := "SrcType := Int" } EQ_Contact(in1 := "DB611".StepDelay."Noof StepsPv", in2 := 9)
   END_RUNG wire#w2
   RUNG wire#w1
      { S7_Templates := "SrcType := Int" } EQ_Contact(in1 := "DB611".StepDelay."Noof StepsPv", in2 := 10)
   END_RUNG wire#w2
   RUNG wire#w1
      { S7_Templates := "SrcType := Int" } EQ_Contact(in1 := "DB611".StepDelay."Noof StepsPv", in2 := 11)
   END_RUNG wire#w2
   RUNG wire#w1
      { S7_Templates := "SrcType := Int" } EQ_Contact(in1 := "DB611".StepDelay."Noof StepsPv", in2 := 16)
   END_RUNG wire#w2
   RUNG wire#w1
      { S7_Templates := "SrcType := Int" } EQ_Contact(in1 := "DB615".CurrentStep, in2 := 9)
   END_RUNG wire#w2
   RUNG wire#w1
      { S7_Templates := "SrcType := Int" } EQ_Contact(in1 := "DB615".CurrentStep, in2 := 10)
   END_RUNG wire#w2
   RUNG wire#w1
      { S7_Templates := "SrcType := Int" } EQ_Contact(in1 := "DB615".CurrentStep, in2 := 11)
   END_RUNG wire#w2
   RUNG wire#w1
      { S7_Templates := "SrcType := Int" } EQ_Contact(in1 := "DB615".CurrentStep, in2 := 15)
   END_RUNG wire#w2
   RUNG wire#w1
      { S7_Templates := "SrcType := Int" } EQ_Contact(in1 := "DB615".CurrentStep, in2 := 16)
   END_RUNG wire#w2
   RUNG wire#w1
      { S7_Templates := "SrcType := Int" } EQ_Contact(in1 := "DB611".StepDelay."Noof StepsPv", in2 := 15)
   END_RUNG wire#w2
   RUNG wire#w1
      { S7_Templates := "SrcType := Int" } EQ_Contact(in1 := "DB611".StepDelay."Noof StepsPv", in2 := 12)
      wire#w3
      { S7_Templates := "[card := 2, value_type := Real]" } MIN(in1 := "AiDb".Ai11.ActValue, in2 := "AiDb".Ai13.ActValue, out => "DB615".ApActPressure)
   END_RUNG
   RUNG wire#w1
      { S7_Templates := "SrcType := Int" } EQ_Contact(in1 := "DB611".StepDelay."Noof StepsPv", in2 := 13)
   END_RUNG wire#w3
   RUNG wire#w1
      { S7_Templates := "SrcType := Int" } EQ_Contact(in1 := "DB611".StepDelay."Noof StepsPv", in2 := 14)
      wire#w4
      { S7_Templates := "[card := 3, value_type := Real]" } MIN(in1 := "AiDb".Ai11.ActValue, in2 := "AiDb".Ai13.ActValue, in3 := "AiDb".Ai14.ActValue, out => "DB615".ApActPressure)
   END_RUNG
   RUNG wire#w1
      { S7_Templates := "SrcType := Int" } EQ_Contact(in1 := "DB611".StepDelay."Noof StepsPv", in2 := 17)
   END_RUNG wire#w4
   RUNG wire#w1
      { S7_Templates := "SrcType := Int" } EQ_Contact(in1 := "DB611".StepDelay."Noof StepsPv", in2 := 6)
      Move(in := "AiDb".Ai12.ActValue, out1 => "DB615".ApActPressure)
   END_RUNG
   // the same network as SCL:
   #_w1 := "AlwaysTRUE" AND "DB615".Selected;
   IF #_w1 AND (("DB611".StepDelay."Noof StepsPv" <= 5) OR ("DB611".StepDelay."Noof StepsPv" = 7) OR ("DB611".StepDelay."Noof StepsPv" = 8) OR ("DB611".StepDelay."Noof StepsPv" = 9) OR ("DB611".StepDelay."Noof StepsPv" = 10) OR ("DB611".StepDelay."Noof StepsPv" = 11) OR ("DB611".StepDelay."Noof StepsPv" = 16) OR ("DB615".CurrentStep = 9) OR ("DB615".CurrentStep = 10) OR ("DB615".CurrentStep = 11) OR ("DB615".CurrentStep = 15) OR ("DB615".CurrentStep = 16) OR ("DB611".StepDelay."Noof StepsPv" = 15)) THEN
       "DB615".ApActPressure := "AiDb".Ai11.ActValue;
   END_IF;
   IF #_w1 AND (("DB611".StepDelay."Noof StepsPv" = 12) OR ("DB611".StepDelay."Noof StepsPv" = 13)) THEN
       "DB615".ApActPressure := MIN(IN1 := "AiDb".Ai11.ActValue, IN2 := "AiDb".Ai13.ActValue);
   END_IF;
   IF #_w1 AND (("DB611".StepDelay."Noof StepsPv" = 14) OR ("DB611".StepDelay."Noof StepsPv" = 17)) THEN
       "DB615".ApActPressure := MIN(IN1 := "AiDb".Ai11.ActValue, IN2 := "AiDb".Ai13.ActValue, IN3 := "AiDb".Ai14.ActValue);
   END_IF;
   IF #_w1 AND ("DB611".StepDelay."Noof StepsPv" = 6) THEN
       "DB615".ApActPressure := "AiDb".Ai12.ActValue;
   END_IF;
END_REGION
END_FUNCTION
